// TIA Portal V17 export
// export: Created 2026-04-12T10:31:16.1811111Z, ExportSetting WithDefaults, DisplayName Totally Integrated Automation Portal, DisplayVersion V17 Update 4, DisplayName TIA Portal Openness, DisplayVersion V17 Update 4, DisplayName TIA Portal Version Control Interface, DisplayVersion V17, DisplayName SINAMICS Startdrive Advanced, DisplayVersion V17, DisplayName SINAMICS Startdrive G130, G150, S120, S150, SINAMICS MV, S210, DisplayVersion V17, DisplayName SINAMICS Startdrive G110M, G120, G120C, G120D, G120P, G115D, DisplayVersion V17, DisplayName STEP 7 Professional, DisplayVersion V17 Update 4, DisplayName STEP 7 Safety, DisplayVersion V17, DisplayName WinCC Advanced, DisplayVersion V17 Update 4
FUNCTION "报警" : Void   // FC5, LAD
{ S7_Optimized_Access := 'TRUE' }
VERSION : 0.1
// stored: AutoNumber true, IsIECCheckEnabled false, SetENOAutomatically false, UDAEnableTagReadback false
   VAR_TEMP   // added for the SCL form of the ladder/FBD networks
      _w1 : Bool;
      _w2 : Bool;
      _w3 : Bool;
      _w4 : Bool;
   END_VAR
BEGIN

REGION Network 1: 控温通讯故障
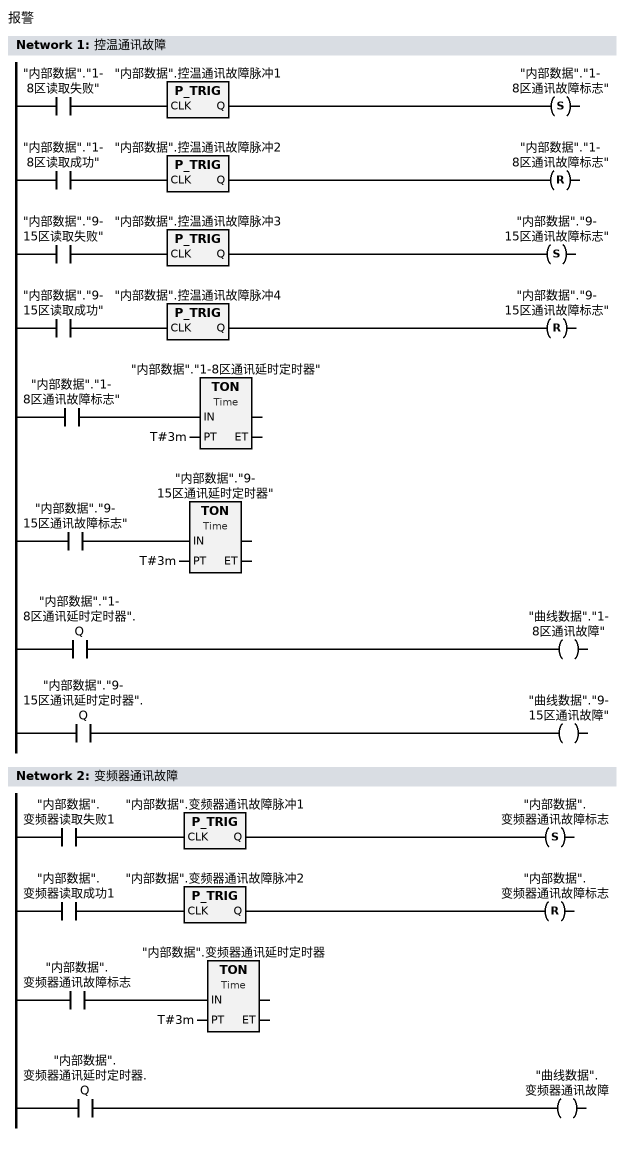
   RUNG wire#powerrail
      Contact( "内部数据"."1-8区读取失败" )
      P_Trig( "内部数据".控温通讯故障脉冲1 )
      S_Coil( "内部数据"."1-8区通讯故障标志" )
   END_RUNG
   RUNG wire#powerrail
      Contact( "内部数据"."1-8区读取成功" )
      P_Trig( "内部数据".控温通讯故障脉冲2 )
      R_Coil( "内部数据"."1-8区通讯故障标志" )
   END_RUNG
   RUNG wire#powerrail
      Contact( "内部数据"."9-15区读取失败" )
      P_Trig( "内部数据".控温通讯故障脉冲3 )
      S_Coil( "内部数据"."9-15区通讯故障标志" )
   END_RUNG
   RUNG wire#powerrail
      Contact( "内部数据"."9-15区读取成功" )
      P_Trig( "内部数据".控温通讯故障脉冲4 )
      R_Coil( "内部数据"."9-15区通讯故障标志" )
   END_RUNG
   RUNG wire#powerrail
      Contact( "内部数据"."1-8区通讯故障标志" )
      { S7_Templates := "time_type := Time" } "内部数据"."1-8区通讯延时定时器".TON(pt := T#3m, et =>)
   END_RUNG
   RUNG wire#powerrail
      Contact( "内部数据"."9-15区通讯故障标志" )
      { S7_Templates := "time_type := Time" } "内部数据"."9-15区通讯延时定时器".TON(pt := T#3m, et =>)
   END_RUNG
   RUNG wire#powerrail
      Contact( "内部数据"."1-8区通讯延时定时器".Q )
      Coil( "曲线数据"."1-8区通讯故障" )
   END_RUNG
   RUNG wire#powerrail
      Contact( "内部数据"."9-15区通讯延时定时器".Q )
      Coil( "曲线数据"."9-15区通讯故障" )
   END_RUNG
   // the same network as SCL:
   #_w1 := "内部数据"."1-8区读取失败" AND NOT "内部数据".控温通讯故障脉冲1;   // rising edge
   "内部数据".控温通讯故障脉冲1 := "内部数据"."1-8区读取失败";
   IF #_w1 THEN "内部数据"."1-8区通讯故障标志" := TRUE; END_IF;
   #_w2 := "内部数据"."1-8区读取成功" AND NOT "内部数据".控温通讯故障脉冲2;   // rising edge
   "内部数据".控温通讯故障脉冲2 := "内部数据"."1-8区读取成功";
   IF #_w2 THEN "内部数据"."1-8区通讯故障标志" := FALSE; END_IF;
   #_w3 := "内部数据"."9-15区读取失败" AND NOT "内部数据".控温通讯故障脉冲3;   // rising edge
   "内部数据".控温通讯故障脉冲3 := "内部数据"."9-15区读取失败";
   IF #_w3 THEN "内部数据"."9-15区通讯故障标志" := TRUE; END_IF;
   #_w4 := "内部数据"."9-15区读取成功" AND NOT "内部数据".控温通讯故障脉冲4;   // rising edge
   "内部数据".控温通讯故障脉冲4 := "内部数据"."9-15区读取成功";
   IF #_w4 THEN "内部数据"."9-15区通讯故障标志" := FALSE; END_IF;
   "内部数据"."1-8区通讯延时定时器".TON(IN := "内部数据"."1-8区通讯故障标志", PT := T#3m);
   "内部数据"."9-15区通讯延时定时器".TON(IN := "内部数据"."9-15区通讯故障标志", PT := T#3m);
   "曲线数据"."1-8区通讯故障" := "内部数据"."1-8区通讯延时定时器".Q;
   "曲线数据"."9-15区通讯故障" := "内部数据"."9-15区通讯延时定时器".Q;
END_REGION

REGION Network 2: 变频器通讯故障
   RUNG wire#powerrail
      Contact( "内部数据".变频器读取失败1 )
      P_Trig( "内部数据".变频器通讯故障脉冲1 )
      S_Coil( "内部数据".变频器通讯故障标志 )
   END_RUNG
   RUNG wire#powerrail
      Contact( "内部数据".变频器读取成功1 )
      P_Trig( "内部数据".变频器通讯故障脉冲2 )
      R_Coil( "内部数据".变频器通讯故障标志 )
   END_RUNG
   RUNG wire#powerrail
      Contact( "内部数据".变频器通讯故障标志 )
      { S7_Templates := "time_type := Time" } "内部数据".变频器通讯延时定时器.TON(pt := T#3m, et =>)
   END_RUNG
   RUNG wire#powerrail
      Contact( "内部数据".变频器通讯延时定时器.Q )
      Coil( "曲线数据".变频器通讯故障 )
   END_RUNG
   // the same network as SCL:
   #_w1 := "内部数据".变频器读取失败1 AND NOT "内部数据".变频器通讯故障脉冲1;   // rising edge
   "内部数据".变频器通讯故障脉冲1 := "内部数据".变频器读取失败1;
   IF #_w1 THEN "内部数据".变频器通讯故障标志 := TRUE; END_IF;
   #_w2 := "内部数据".变频器读取成功1 AND NOT "内部数据".变频器通讯故障脉冲2;   // rising edge
   "内部数据".变频器通讯故障脉冲2 := "内部数据".变频器读取成功1;
   IF #_w2 THEN "内部数据".变频器通讯故障标志 := FALSE; END_IF;
   "内部数据".变频器通讯延时定时器.TON(IN := "内部数据".变频器通讯故障标志, PT := T#3m);
   "曲线数据".变频器通讯故障 := "内部数据".变频器通讯延时定时器.Q;
END_REGION
END_FUNCTION
